FUNCTION_BLOCK F_EXPN (* calculates X to the power of N (Y = X^N) *)
  (* Standard: OSCAT; Classification: Math *)
  (* Version 0.0, 2011-07-21, 4DIAC-IDE, 4DIAC-Consortium *)
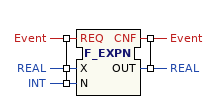
  EVENT_INPUT
    REQ WITH X, N; (* Service Request *)
  END_EVENT
  EVENT_OUTPUT
    CNF WITH OUT; (* Confirmation of Requested Service *)
  END_EVENT
  VAR_INPUT
    X : REAL; (* Input *)
    N : INT; (* Exponential *)
  END_VAR
  VAR_OUTPUT
    OUT : REAL; (* Outcome *)
  END_VAR
END_FUNCTION_BLOCK
